FUNCTION_BLOCK FB_SEW_MovidriveB EXTENDS FB_BaseDevice

VAR_INPUT 
	// PA2 + PA3 TARGET POSITION
	nTargetPosition: DINT;  // User defined units
	// PA4: SETPOINT SPEED
	nSetpointSpeed: INT; // 1/min
	// PA5 + PA6: ACCELERATION RAMP AND DECELERATION RAMP
	tRamp_Accel: TIME; // 16-bit INT - in seconds
	tRamp_Decel: TIME; // 16-bit INT - in seconds
END_VAR


VAR_OUTPUT
	// PE2 + PE3 ACTUAL POSITION
	nActualPosition: DINT;  // User defined units
	//PE4: ACTUAL SPEED
	nActualSpeed: INT; // 1/min
	//PE5: ACTIVE CURRENT
	nActiveCurrent: INT; // % of rated current
	//PE6: UNIT UTILISATION
	nUnitUtilisation: INT; // % I x t
END_VAR

VAR
	// PROCESS OUTPUT DATA 
	// PO1: CONTROL WORD 2
	bSWLimitSwitch: BOOL;
	bModeHigh: BOOL;
	bModeLow: BOOL;
	bJog_Rev: BOOL := FALSE;
	bJog_Fwd: BOOL := FALSE;
	bStart: BOOL;
	bFaultReset: BOOL;
	bParamSet_SwitchOver: BOOL;
	bRampSwitchover: BOOL;
	bHold_Ctrl: BOOL;
	bEnable_Stop: BOOL;
	bEnable_RapidStop: BOOL;
	bController_Inhibit: BOOL;

	//PROCESS INPUT DATA
	
	// PE1 STATUS WORD
	FaultCode: BYTE;
	bLimSwitch_CCW: BOOL;
	bLimSwitch_CW: BOOL;
	bFault: BOOL;
	bBrakeReleased: BOOL;
	bTargetPosReached: BOOL;
	bIPOSReference: BOOL;
	bInverterReady: BOOL;
	bMotorTurning: BOOL;
	
	// PROCESS DATA WORDS to LINK TO DRIVE
	PO1_ProcessOutput_1 AT %Q* : WORD;
	PO2_ProcessOutput_2 AT %Q* : WORD;
	PO3_ProcessOutput_3 AT %Q* : WORD;
	PO4_ProcessOutput_4 AT %Q* : WORD;
	PO5_ProcessOutput_5 AT %Q* : WORD;
	PO6_ProcessOutput_6 AT %Q* : WORD;
	
	PI1_ProcessInput_1 AT %I* : WORD;
	PI2_ProcessInput_2 AT %I* : WORD;
	PI3_ProcessInput_3 AT %I* : WORD;
	PI4_ProcessInput_4 AT %I* : WORD;
	PI5_ProcessInput_5 AT %I* : WORD;
	PI6_ProcessInput_6 AT %I* : WORD;
	
	// Additional Variables
	eOperatingMode: E_MovidriveB_OpMode := E_MovidriveB_OpMode.JOG_MODE;
	
END_VAR

VAR_OUTPUT PERSISTENT 
	bExtending_1_or_Retracting_0: BOOL;
END_VAR

VAR PERSISTENT
	bAbove_1_or_Below_0_HomePos: BOOL;
	eSMState: (INIT, ENABLE, REFEREN, MOVE_TRIG, MOVING, MOVED, STOP, ERROR, RESET) := INIT;
	nGearRation: REAL; 
	nInertia: REAL;
END_VAR

updateInputs();
updateOutputs();


IF nActualPosition > 0 THEN
	bAbove_1_or_Below_0_HomePos := TRUE;
ELSE
	bAbove_1_or_Below_0_HomePos := FALSE;
END_IF

IF eStateTarget = E_DeviceState.EXTENDED THEN
	eSMState := MOVE_TRIG;
END_IF


CASE eSMState OF
	INIT:
		bController_Inhibit := TRUE;
		bHold_Ctrl := TRUE;
		
	ENABLE:
		bController_Inhibit := FALSE;
		bHold_Ctrl := FALSE;
		eState := E_DeviceState.IDLE;
		bStart := FALSE;
		bEnable_Stop := TRUE;
		bEnable_RapidStop := TRUE;
		
	REFEREN:
			bModeLow 	:= FALSE;
			bModeHigh 	:= TRUE;
			bStart := TRUE;
	
	MOVE_TRIG:
		IF bInverterReady AND ( NOT bFault ) THEN
			bModeLow 	:= TRUE;
			bModeHigh 	:= TRUE;
			eSMState := MOVING;
			
			IF nActualPosition < nTargetPosition THEN
				bExtending_1_or_Retracting_0 := TRUE;
			ELSE
				bExtending_1_or_Retracting_0 := FALSE;
			END_IF
			
		ELSE
			eSMState := ERROR;
		END_IF
		
	MOVING:
		eState := E_DeviceState.EXTENDING;
		bStart := TRUE;
		IF bTargetPosReached THEN
			eSMState := MOVED;
		END_IF
		
	MOVED:
		eState := E_DeviceState.EXTENDED;
		eSMState := ENABLE;
		bStart := FALSE;
		
	STOP:
		bEnable_Stop := TRUE;
			
	
	ERROR:
		IF bFault THEN
			CASE FaultCode OF
				07:
					// Under-voltage
				08:
					// N-monitoring
				10:
					// IPOS-ILLOP
				14:
					// Encoder
				25:
					// EEPROM
				28:
					// Field-bus timeout
				29:
					// Limit switch reached
				31: 
					// TF Sensor
				36:
					// Immediate switch-off
				42: 
					// Lag fault
				94: 
					// EEPROM checksum
			END_CASE
		END_IF
		//
	RESET:
		bFaultReset := TRUE;
		//
END_CASE

METHOD updateInputs : BOOL
VAR_INPUT
END_VAR
FaultCode 			:= INT_TO_BYTE(SHR((PI1_ProcessInput_1 AND 16#F0), 8));
bLimSwitch_CCW 		:= PI1_ProcessInput_1.7;
bLimSwitch_CW 		:= PI1_ProcessInput_1.6;
bFault 				:= PI1_ProcessInput_1.5;
bBrakeReleased		:= PI1_ProcessInput_1.4;
bTargetPosReached 	:= PI1_ProcessInput_1.3;
bIPOSReference 		:= PI1_ProcessInput_1.2;
bInverterReady 		:= PI1_ProcessInput_1.1;
bMotorTurning 		:= PI1_ProcessInput_1.0;
nActualPosition 	:= SHL(WORD_TO_DWORD(PI2_ProcessInput_2), 16) OR WORD_TO_DWORD(PI3_ProcessInput_3);
nActualSpeed 		:= WORD_TO_INT(PI4_ProcessInput_4);
nActiveCurrent 		:= WORD_TO_INT(PI5_ProcessInput_5);
nUnitUtilisation 	:= WORD_TO_INT(PI6_ProcessInput_6);
END_METHOD

METHOD updateOutputs : BOOL
VAR_INPUT
END_VAR
PO1_ProcessOutput_1.15 := bSWLimitSwitch;
PO1_ProcessOutput_1.12 := bModeHigh;
PO1_ProcessOutput_1.11 := bModeLow;
PO1_ProcessOutput_1.10 := bJog_Rev;
PO1_ProcessOutput_1.9 := bJog_Fwd;
PO1_ProcessOutput_1.8 := bStart;
PO1_ProcessOutput_1.6 := bFaultReset;
PO1_ProcessOutput_1.5 := bParamSet_SwitchOver;
PO1_ProcessOutput_1.4 := bRampSwitchover;
PO1_ProcessOutput_1.3 := bHold_Ctrl;
PO1_ProcessOutput_1.2 := bEnable_Stop; 
PO1_ProcessOutput_1.1 := bEnable_RapidStop;
PO1_ProcessOutput_1.0 := bController_Inhibit;

PO2_ProcessOutput_2 := DINT_TO_WORD(SHR(nTargetPosition AND 2#11111111111111110000000000000000, 16));
PO3_ProcessOutput_3 := UDINT_TO_WORD(nTargetPosition AND 2#1111111111111111);

PO4_ProcessOutput_4 := INT_TO_WORD(nSetpointSpeed);

PO5_ProcessOutput_5 := DINT_TO_WORD(TIME_TO_DINT(tRamp_Accel));
PO6_ProcessOutput_6 := DINT_TO_WORD(TIME_TO_DINT(tRamp_Decel));
END_METHOD

END_FUNCTION_BLOCK

(* stored: Version 1.1.0.1, ProductVersion 3.1.4024.12
   POU FB_SEW_MovidriveB: Id {15081331-1a1c-4e92-b26a-deb052c11093}, SpecialFunc None
   Method updateInputs: Id {85468d3e-1cca-4dc0-8611-e08853e4d66e}
   Method updateOutputs: Id {d717cb8f-1931-401b-8aac-06bb4ded51d8} *)
